(* CoDeSys 2.3.9.62 project: AscensorCompletoDobleV1-2.pro *)
(* Libraries: Standard.lib 2.6.14 10:37:46, IecSfc.lib 2.6.14 12:37:46 *)

(* Global variable list: Global_Variables *)
VAR_GLOBAL
   (*Entradas *)
      (* Sensores de posición en plantas *)
      S0_1: BOOL;
      S1_1: BOOL;
      S2_1: BOOL;
      S3_1: BOOL;
      S0_2: BOOL;
      S1_2: BOOL;
      S2_2: BOOL;
      S3_2: BOOL;
      (* Pulsadores de llamadas en planta *)
      P0: BOOL;
      P1: BOOL;
      P2: BOOL;
      P3: BOOL;
    (* Pulsadores en cabina  *)
      C0_1: BOOL;
      C1_1: BOOL;
      C2_1: BOOL;
      C3_1: BOOL;
      C0_2: BOOL;
      C1_2: BOOL;
      C2_2: BOOL;
      C3_2: BOOL;
   (*Salidas *)
      Motor_arriba_1 : BOOL;
      Motor_Abajo_1 : BOOL;
     Motor_arriba_2 : BOOL;
      Motor_Abajo_2 : BOOL;
   (* luces asociadas a los pulsadores. Se usarán
        si se quiere implementar memoria de llamada *)
     LuzP0:BOOL;
     LuzP1:BOOL;
     LuzP2:BOOL;
     LuzP3:BOOL;
     LuzC0_1:BOOL;
     LuzC1_1:BOOL;
     LuzC2_1:BOOL;
     LuzC3_1:BOOL;
     LuzC0_2:BOOL;
     LuzC1_2:BOOL;
     LuzC2_2:BOOL;
     LuzC3_2:BOOL;
END_VAR

(* POU PLC_PRG, ST *)
PROGRAM PLC_PRG
VAR
	memoria11 : INT := 0;
	memoria12 : INT := 0;
	memoria13 : INT  :=0;
END_VAR
Movimiento1;
Movimiento2;

(* Ascensor 1 *)
Ascensor1;
END_PROGRAM

(* POU Movimiento1, ST *)
PROGRAM Movimiento1
VAR
    pos1:INT:=0;
END_VAR
IF (Motor_arriba_1 AND pos1>=-240) THEN
   pos1:=pos1-2;
END_IF


IF (Motor_abajo_1 AND pos1<=-2) THEN
   pos1:=pos1+2;
END_IF

IF (pos1>=0 AND pos1<=2) THEN
  S0_1:=TRUE;
ELSE
  S0_1:=FALSE;
END_IF

IF (pos1>=-78 AND pos1<=-74) THEN
  S1_1:=TRUE;
ELSE
  S1_1:=FALSE;
END_IF

IF (pos1>=-156 AND pos1<=-152) THEN
  S2_1:=TRUE;
ELSE
  S2_1:=FALSE;
END_IF

IF (pos1>=-242 AND pos1<=-240) THEN
  S3_1:=TRUE;
ELSE
  S3_1:=FALSE;
END_IF
END_PROGRAM

(* POU Movimiento2, ST *)
PROGRAM Movimiento2
VAR
    pos2:INT:=0;
END_VAR
IF (Motor_arriba_2 AND pos2>=-240) THEN
   pos2:=pos2-2;
END_IF


IF (Motor_abajo_2 AND pos2<=-2) THEN
   pos2:=pos2+2;
END_IF

IF (pos2>=0 AND pos2<=2) THEN
  S0_2:=TRUE;
ELSE
  S0_2:=FALSE;
END_IF

IF (pos2>=-78 AND pos2<=-74) THEN
  S1_2:=TRUE;
ELSE
  S1_2:=FALSE;
END_IF

IF (pos2>=-156 AND pos2<=-152) THEN
  S2_2:=TRUE;
ELSE
  S2_2:=FALSE;
END_IF

IF (pos2>=-242 AND pos2<=-240) THEN
  S3_2:=TRUE;
ELSE
  S3_2:=FALSE;
END_IF
END_PROGRAM

(* POU Ascensor1, LD *)
PROGRAM Ascensor1
VAR
	Parado1: BOOL;
	Marcha1: BOOL;
	Sube1_12: BOOL;
	Sube1_01: BOOL;
	Sube1_02: BOOL;
	Sube1_03: BOOL;
	Baja1_10: BOOL;
	Sube1_13: BOOL;
	Baja1_20: BOOL;
	Baja1_21: BOOL;
	Sube1_23: BOOL;
	Baja1_30: BOOL;
	Baja1_31: BOOL;
	Baja1_32: BOOL;
	Marcha2: BOOL;
	Sube2_01: BOOL;
	Sube2_02: BOOL;
	Sube2_03: BOOL;
	Baja2_10: BOOL;
	Sube2_12: BOOL;
	Sube2_13: BOOL;
	Baja2_20: BOOL;
	Baja2_21: BOOL;
	Sube2_23: BOOL;
	Baja2_30: BOOL;
	Baja2_31: BOOL;
	Baja2_32: BOOL;
	FIN: BOOL;
END_VAR
VAR (* helpers for the ST form of the networks *)
	_p1 : BOOL;
	_p2 : BOOL;
	_p3 : BOOL;
	_p4 : BOOL;
	_p5 : BOOL;
	_p6 : BOOL;
	_p7 : BOOL;
	_p8 : BOOL;
	_p9 : BOOL;
	_p10 : BOOL;
	_p11 : BOOL;
	_p12 : BOOL;
	_p13 : BOOL;
	_p14 : BOOL;
	_p15 : BOOL;
	_p16 : BOOL;
	_p17 : BOOL;
	_p18 : BOOL;
	_p19 : BOOL;
	_p20 : BOOL;
	_p21 : BOOL;
	_p22 : BOOL;
	_p23 : BOOL;
	_p24 : BOOL;
	_p25 : BOOL;
	_p26 : BOOL;
	_p27 : BOOL;
	_p28 : BOOL;
	_p29 : BOOL;
	_p30 : BOOL;
	_p31 : BOOL;
	_p32 : BOOL;
	_p33 : BOOL;
	_p34 : BOOL;
	_p35 : BOOL;
	_p36 : BOOL;
	_p37 : BOOL;
	_p38 : BOOL;
	_p39 : BOOL;
	_p40 : BOOL;
	_p41 : BOOL;
	_p42 : BOOL;
	_p43 : BOOL;
	_p44 : BOOL;
	_p45 : BOOL;
	_p46 : BOOL;
	_p47 : BOOL;
	_p48 : BOOL;
	_p49 : BOOL;
	_p50 : BOOL;
	_p51 : BOOL;
	_p52 : BOOL;
	_p53 : BOOL;
	_p54 : BOOL;
	_p55 : BOOL;
	_p56 : BOOL;
	_p57 : BOOL;
	_p58 : BOOL;
	_p59 : BOOL;
	_p60 : BOOL;
	_p61 : BOOL;
	_p62 : BOOL;
END_VAR
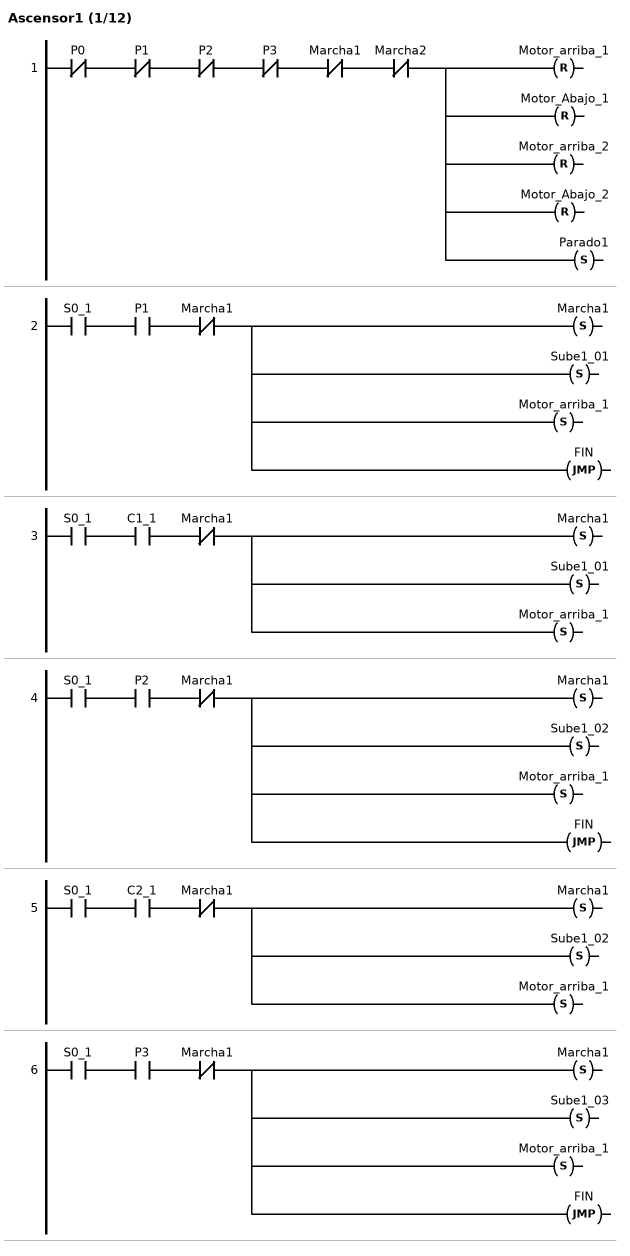
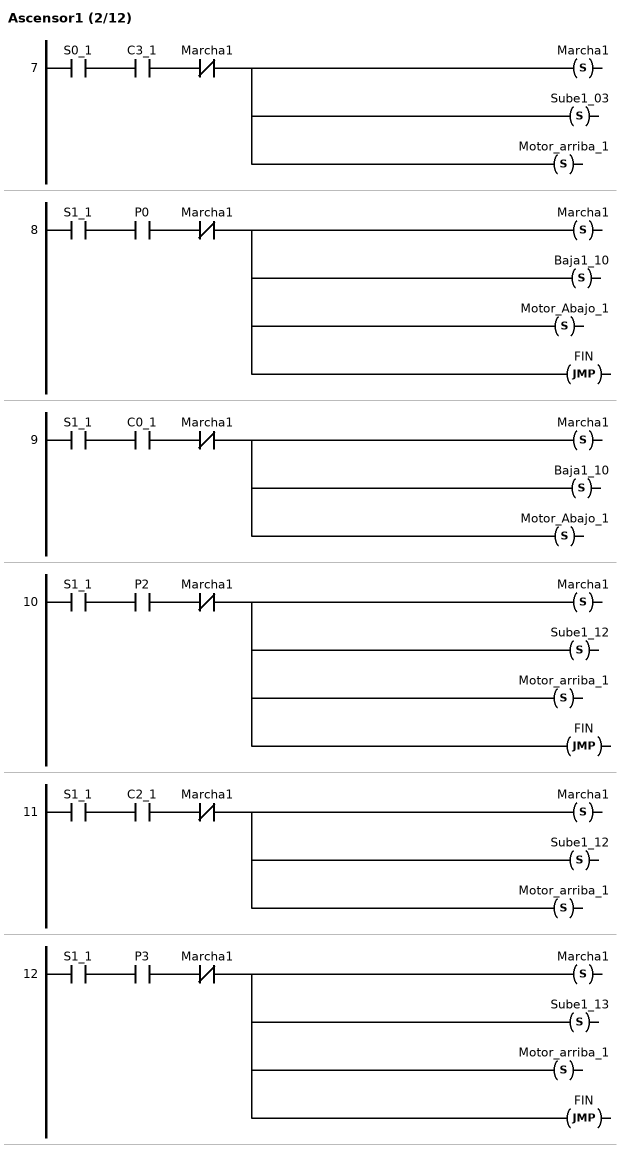
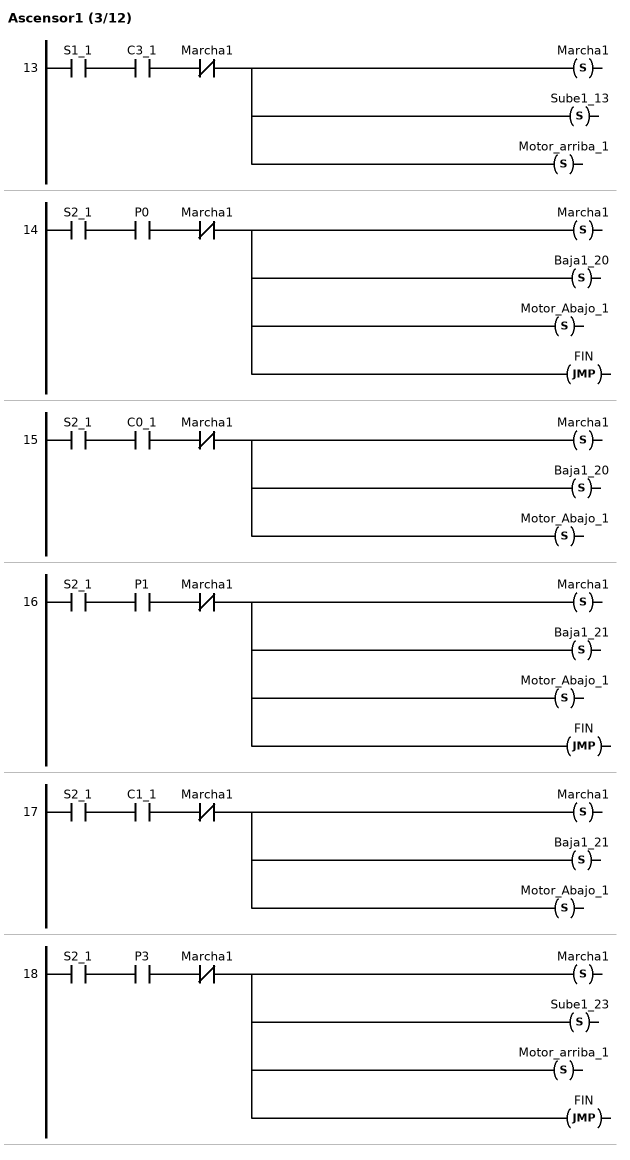
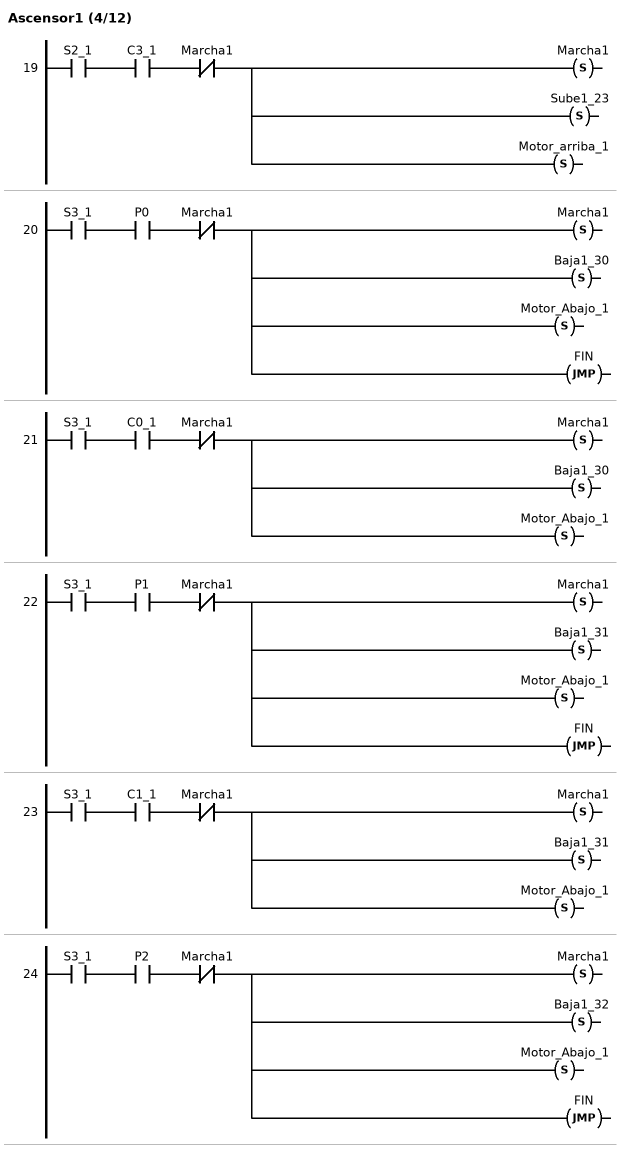
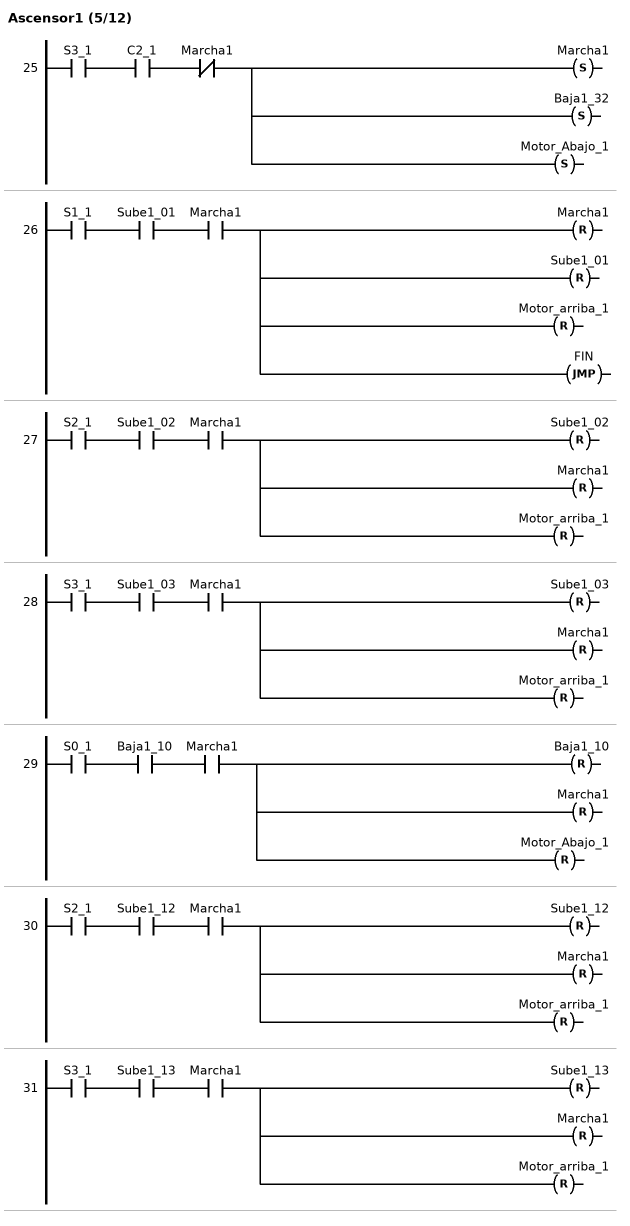
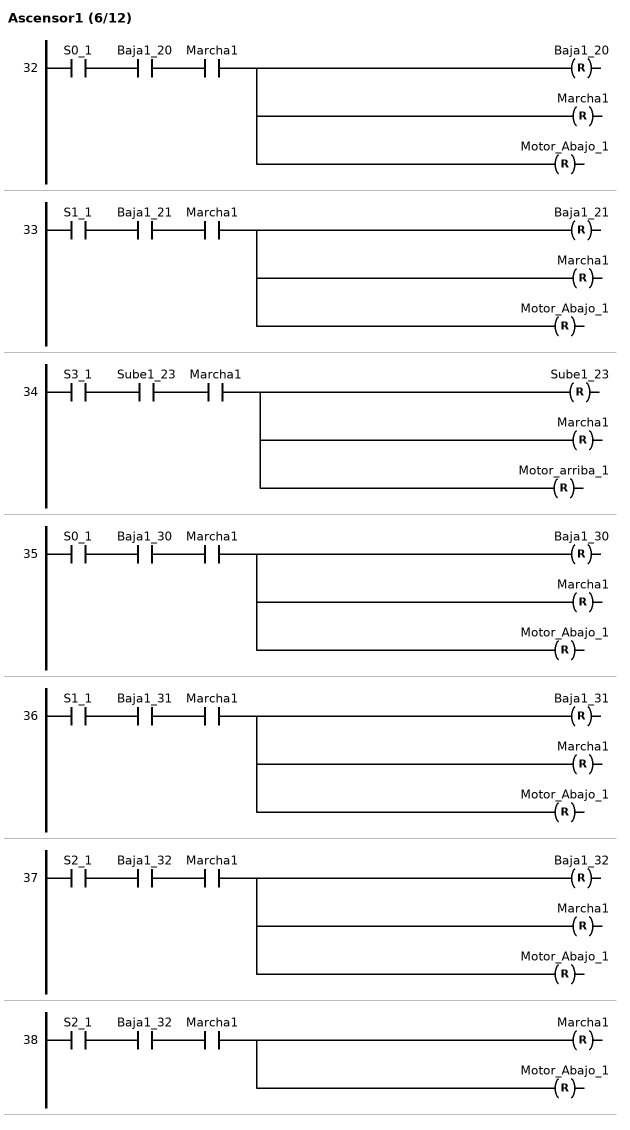
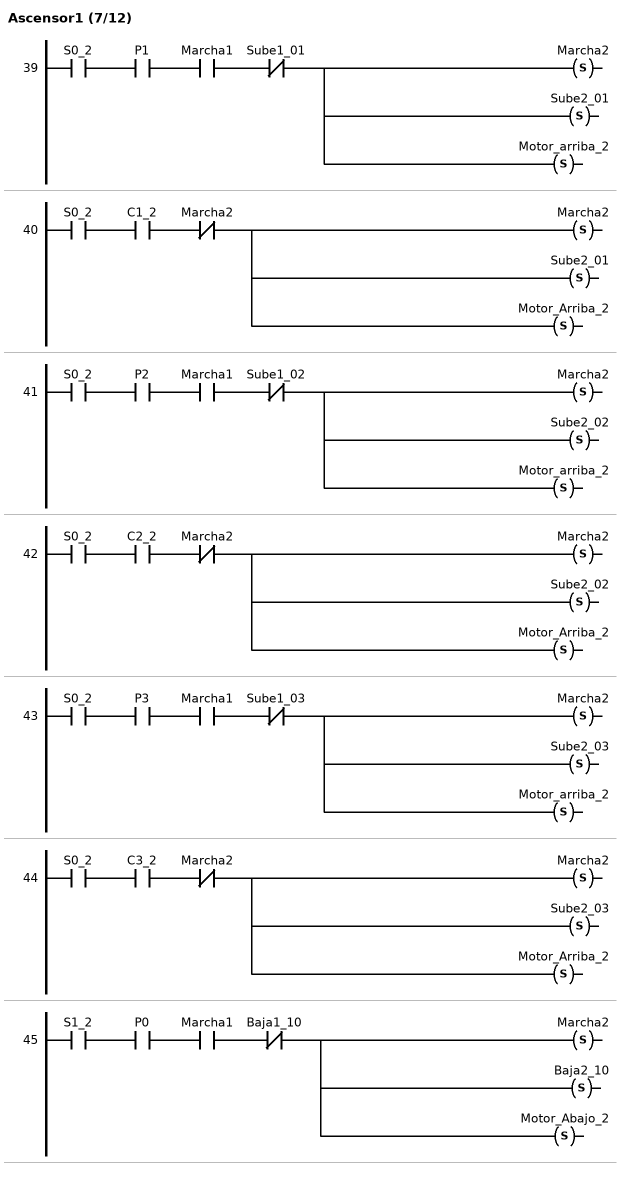
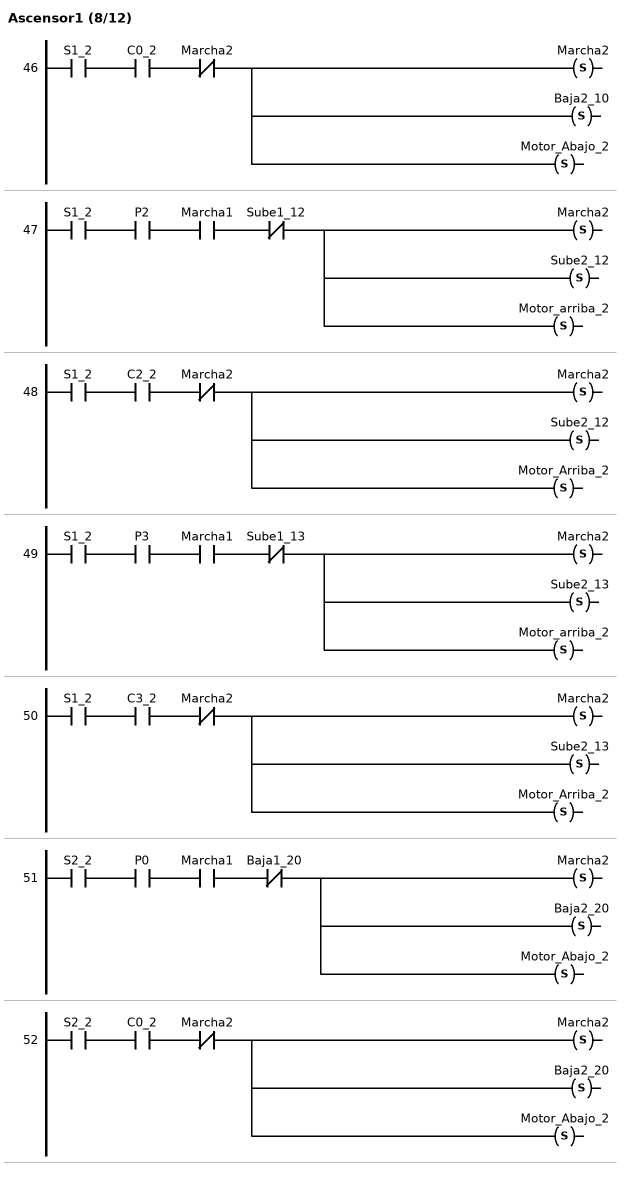
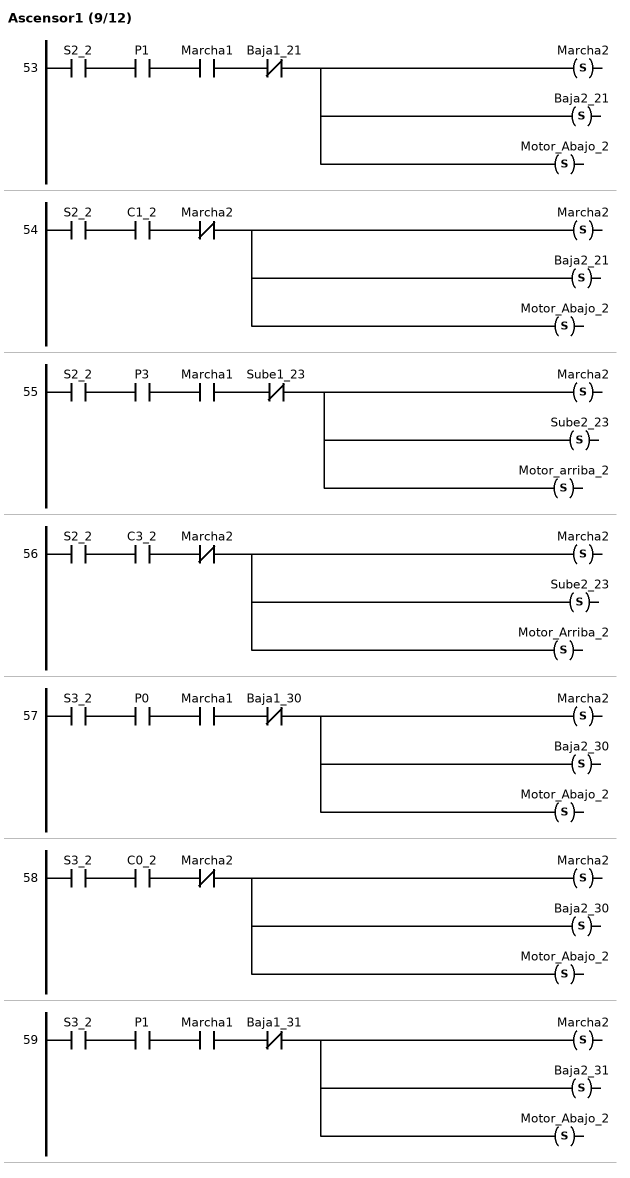
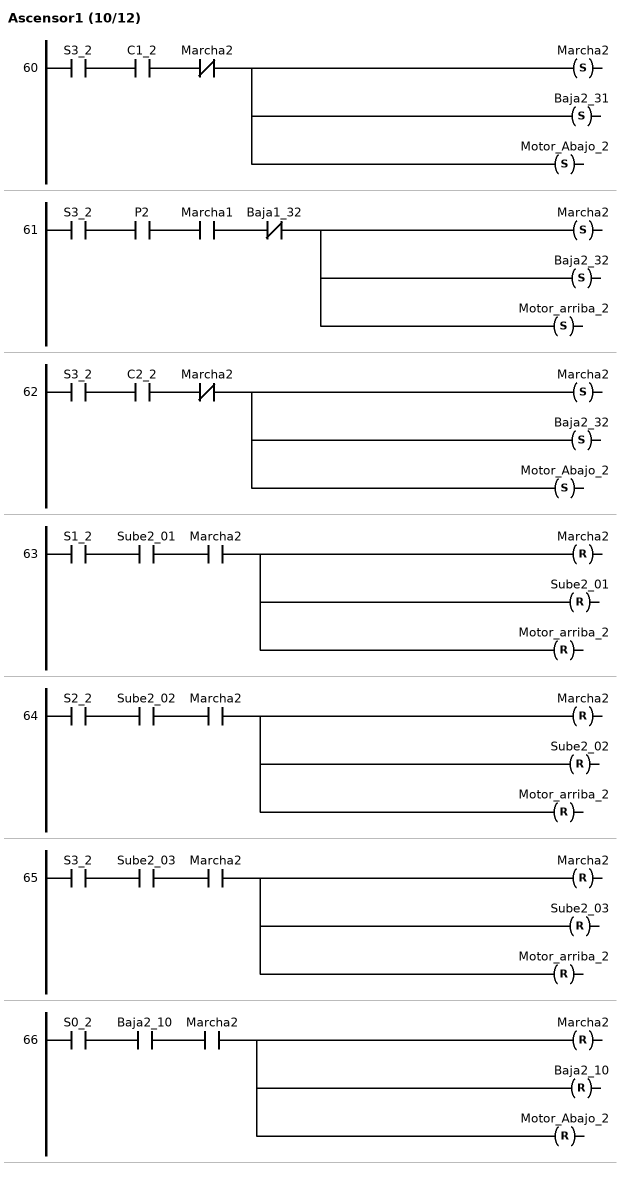
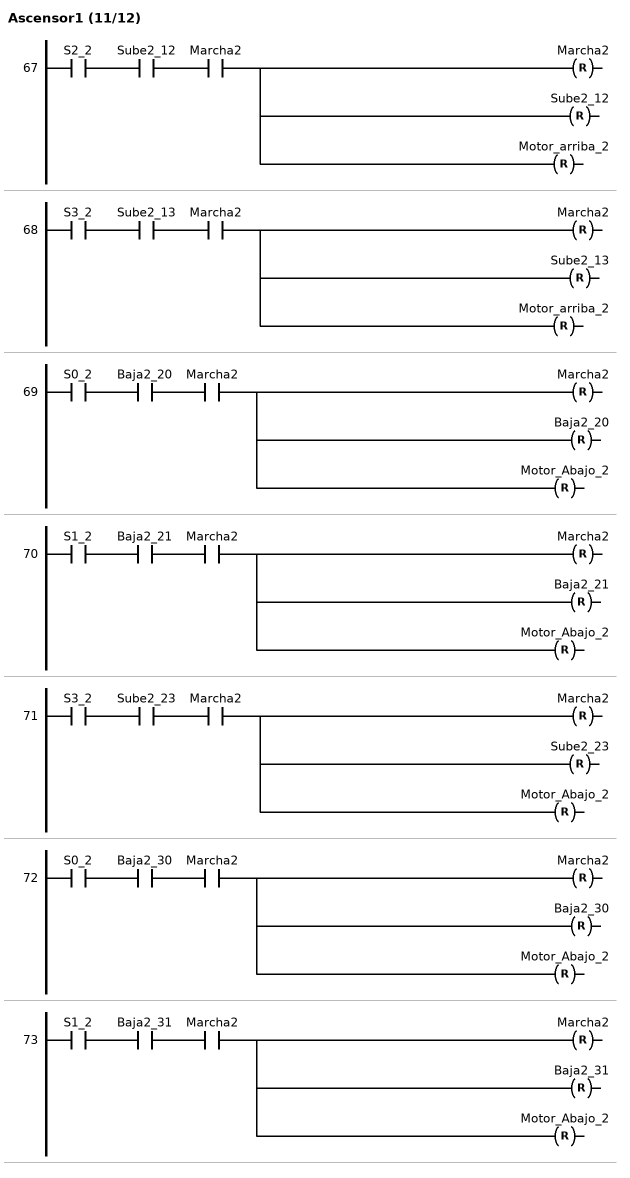
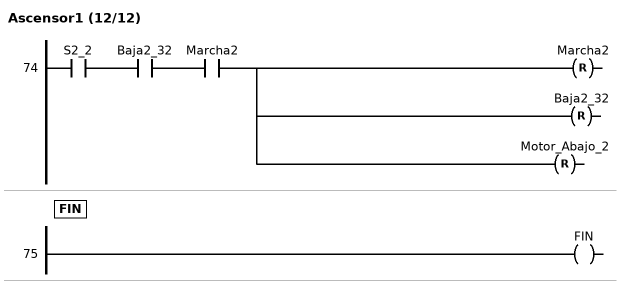
_LD_ (* Ladder Diagram *)
NETWORK 1
	[/P0] - [/P1] - [/P2] - [/P3] - [/Marcha1] - [/Marcha2] --- (R Motor_arriba_1) (R Motor_Abajo_1) (R Motor_arriba_2) (R Motor_Abajo_2) (S Parado1)
NETWORK 2
	[S0_1] - [P1] - [/Marcha1] --- (S Marcha1) (S Sube1_01) (S Motor_arriba_1) >>FIN
NETWORK 3
	[S0_1] - [C1_1] - [/Marcha1] --- (S Marcha1) (S Sube1_01) (S Motor_arriba_1)
NETWORK 4
	[S0_1] - [P2] - [/Marcha1] --- (S Marcha1) (S Sube1_02) (S Motor_arriba_1) >>FIN
NETWORK 5
	[S0_1] - [C2_1] - [/Marcha1] --- (S Marcha1) (S Sube1_02) (S Motor_arriba_1)
NETWORK 6
	[S0_1] - [P3] - [/Marcha1] --- (S Marcha1) (S Sube1_03) (S Motor_arriba_1) >>FIN
NETWORK 7
	[S0_1] - [C3_1] - [/Marcha1] --- (S Marcha1) (S Sube1_03) (S Motor_arriba_1)
NETWORK 8
	[S1_1] - [P0] - [/Marcha1] --- (S Marcha1) (S Baja1_10) (S Motor_Abajo_1) >>FIN
NETWORK 9
	[S1_1] - [C0_1] - [/Marcha1] --- (S Marcha1) (S Baja1_10) (S Motor_Abajo_1)
NETWORK 10
	[S1_1] - [P2] - [/Marcha1] --- (S Marcha1) (S Sube1_12) (S Motor_arriba_1) >>FIN
NETWORK 11
	[S1_1] - [C2_1] - [/Marcha1] --- (S Marcha1) (S Sube1_12) (S Motor_arriba_1)
NETWORK 12
	[S1_1] - [P3] - [/Marcha1] --- (S Marcha1) (S Sube1_13) (S Motor_arriba_1) >>FIN
NETWORK 13
	[S1_1] - [C3_1] - [/Marcha1] --- (S Marcha1) (S Sube1_13) (S Motor_arriba_1)
NETWORK 14
	[S2_1] - [P0] - [/Marcha1] --- (S Marcha1) (S Baja1_20) (S Motor_Abajo_1) >>FIN
NETWORK 15
	[S2_1] - [C0_1] - [/Marcha1] --- (S Marcha1) (S Baja1_20) (S Motor_Abajo_1)
NETWORK 16
	[S2_1] - [P1] - [/Marcha1] --- (S Marcha1) (S Baja1_21) (S Motor_Abajo_1) >>FIN
NETWORK 17
	[S2_1] - [C1_1] - [/Marcha1] --- (S Marcha1) (S Baja1_21) (S Motor_Abajo_1)
NETWORK 18
	[S2_1] - [P3] - [/Marcha1] --- (S Marcha1) (S Sube1_23) (S Motor_arriba_1) >>FIN
NETWORK 19
	[S2_1] - [C3_1] - [/Marcha1] --- (S Marcha1) (S Sube1_23) (S Motor_arriba_1)
NETWORK 20
	[S3_1] - [P0] - [/Marcha1] --- (S Marcha1) (S Baja1_30) (S Motor_Abajo_1) >>FIN
NETWORK 21
	[S3_1] - [C0_1] - [/Marcha1] --- (S Marcha1) (S Baja1_30) (S Motor_Abajo_1)
NETWORK 22
	[S3_1] - [P1] - [/Marcha1] --- (S Marcha1) (S Baja1_31) (S Motor_Abajo_1) >>FIN
NETWORK 23
	[S3_1] - [C1_1] - [/Marcha1] --- (S Marcha1) (S Baja1_31) (S Motor_Abajo_1)
NETWORK 24
	[S3_1] - [P2] - [/Marcha1] --- (S Marcha1) (S Baja1_32) (S Motor_Abajo_1) >>FIN
NETWORK 25
	[S3_1] - [C2_1] - [/Marcha1] --- (S Marcha1) (S Baja1_32) (S Motor_Abajo_1)
NETWORK 26
	[S1_1] - [Sube1_01] - [Marcha1] --- (R Marcha1) (R Sube1_01) (R Motor_arriba_1) >>FIN
NETWORK 27
	[S2_1] - [Sube1_02] - [Marcha1] --- (R Sube1_02) (R Marcha1) (R Motor_arriba_1)
NETWORK 28
	[S3_1] - [Sube1_03] - [Marcha1] --- (R Sube1_03) (R Marcha1) (R Motor_arriba_1)
NETWORK 29
	[S0_1] - [Baja1_10] - [Marcha1] --- (R Baja1_10) (R Marcha1) (R Motor_Abajo_1)
NETWORK 30
	[S2_1] - [Sube1_12] - [Marcha1] --- (R Sube1_12) (R Marcha1) (R Motor_arriba_1)
NETWORK 31
	[S3_1] - [Sube1_13] - [Marcha1] --- (R Sube1_13) (R Marcha1) (R Motor_arriba_1)
NETWORK 32
	[S0_1] - [Baja1_20] - [Marcha1] --- (R Baja1_20) (R Marcha1) (R Motor_Abajo_1)
NETWORK 33
	[S1_1] - [Baja1_21] - [Marcha1] --- (R Baja1_21) (R Marcha1) (R Motor_Abajo_1)
NETWORK 34
	[S3_1] - [Sube1_23] - [Marcha1] --- (R Sube1_23) (R Marcha1) (R Motor_arriba_1)
NETWORK 35
	[S0_1] - [Baja1_30] - [Marcha1] --- (R Baja1_30) (R Marcha1) (R Motor_Abajo_1)
NETWORK 36
	[S1_1] - [Baja1_31] - [Marcha1] --- (R Baja1_31) (R Marcha1) (R Motor_Abajo_1)
NETWORK 37
	[S2_1] - [Baja1_32] - [Marcha1] --- (R Baja1_32) (R Marcha1) (R Motor_Abajo_1)
NETWORK 38
	[S2_1] - [Baja1_32] - [Marcha1] --- (R Marcha1) (R Motor_Abajo_1)
NETWORK 39
	[S0_2] - [P1] - [Marcha1] - [/Sube1_01] --- (S Marcha2) (S Sube2_01) (S Motor_arriba_2)
NETWORK 40
	[S0_2] - [C1_2] - [/Marcha2] --- (S Marcha2) (S Sube2_01) (S Motor_Arriba_2)
NETWORK 41
	[S0_2] - [P2] - [Marcha1] - [/Sube1_02] --- (S Marcha2) (S Sube2_02) (S Motor_arriba_2)
NETWORK 42
	[S0_2] - [C2_2] - [/Marcha2] --- (S Marcha2) (S Sube2_02) (S Motor_Arriba_2)
NETWORK 43
	[S0_2] - [P3] - [Marcha1] - [/Sube1_03] --- (S Marcha2) (S Sube2_03) (S Motor_arriba_2)
NETWORK 44
	[S0_2] - [C3_2] - [/Marcha2] --- (S Marcha2) (S Sube2_03) (S Motor_Arriba_2)
NETWORK 45
	[S1_2] - [P0] - [Marcha1] - [/Baja1_10] --- (S Marcha2) (S Baja2_10) (S Motor_Abajo_2)
NETWORK 46
	[S1_2] - [C0_2] - [/Marcha2] --- (S Marcha2) (S Baja2_10) (S Motor_Abajo_2)
NETWORK 47
	[S1_2] - [P2] - [Marcha1] - [/Sube1_12] --- (S Marcha2) (S Sube2_12) (S Motor_arriba_2)
NETWORK 48
	[S1_2] - [C2_2] - [/Marcha2] --- (S Marcha2) (S Sube2_12) (S Motor_Arriba_2)
NETWORK 49
	[S1_2] - [P3] - [Marcha1] - [/Sube1_13] --- (S Marcha2) (S Sube2_13) (S Motor_arriba_2)
NETWORK 50
	[S1_2] - [C3_2] - [/Marcha2] --- (S Marcha2) (S Sube2_13) (S Motor_Arriba_2)
NETWORK 51
	[S2_2] - [P0] - [Marcha1] - [/Baja1_20] --- (S Marcha2) (S Baja2_20) (S Motor_Abajo_2)
NETWORK 52
	[S2_2] - [C0_2] - [/Marcha2] --- (S Marcha2) (S Baja2_20) (S Motor_Abajo_2)
NETWORK 53
	[S2_2] - [P1] - [Marcha1] - [/Baja1_21] --- (S Marcha2) (S Baja2_21) (S Motor_Abajo_2)
NETWORK 54
	[S2_2] - [C1_2] - [/Marcha2] --- (S Marcha2) (S Baja2_21) (S Motor_Abajo_2)
NETWORK 55
	[S2_2] - [P3] - [Marcha1] - [/Sube1_23] --- (S Marcha2) (S Sube2_23) (S Motor_arriba_2)
NETWORK 56
	[S2_2] - [C3_2] - [/Marcha2] --- (S Marcha2) (S Sube2_23) (S Motor_Arriba_2)
NETWORK 57
	[S3_2] - [P0] - [Marcha1] - [/Baja1_30] --- (S Marcha2) (S Baja2_30) (S Motor_Abajo_2)
NETWORK 58
	[S3_2] - [C0_2] - [/Marcha2] --- (S Marcha2) (S Baja2_30) (S Motor_Abajo_2)
NETWORK 59
	[S3_2] - [P1] - [Marcha1] - [/Baja1_31] --- (S Marcha2) (S Baja2_31) (S Motor_Abajo_2)
NETWORK 60
	[S3_2] - [C1_2] - [/Marcha2] --- (S Marcha2) (S Baja2_31) (S Motor_Abajo_2)
NETWORK 61
	[S3_2] - [P2] - [Marcha1] - [/Baja1_32] --- (S Marcha2) (S Baja2_32) (S Motor_arriba_2)
NETWORK 62
	[S3_2] - [C2_2] - [/Marcha2] --- (S Marcha2) (S Baja2_32) (S Motor_Abajo_2)
NETWORK 63
	[S1_2] - [Sube2_01] - [Marcha2] --- (R Marcha2) (R Sube2_01) (R Motor_arriba_2)
NETWORK 64
	[S2_2] - [Sube2_02] - [Marcha2] --- (R Marcha2) (R Sube2_02) (R Motor_arriba_2)
NETWORK 65
	[S3_2] - [Sube2_03] - [Marcha2] --- (R Marcha2) (R Sube2_03) (R Motor_arriba_2)
NETWORK 66
	[S0_2] - [Baja2_10] - [Marcha2] --- (R Marcha2) (R Baja2_10) (R Motor_Abajo_2)
NETWORK 67
	[S2_2] - [Sube2_12] - [Marcha2] --- (R Marcha2) (R Sube2_12) (R Motor_arriba_2)
NETWORK 68
	[S3_2] - [Sube2_13] - [Marcha2] --- (R Marcha2) (R Sube2_13) (R Motor_arriba_2)
NETWORK 69
	[S0_2] - [Baja2_20] - [Marcha2] --- (R Marcha2) (R Baja2_20) (R Motor_Abajo_2)
NETWORK 70
	[S1_2] - [Baja2_21] - [Marcha2] --- (R Marcha2) (R Baja2_21) (R Motor_Abajo_2)
NETWORK 71
	[S3_2] - [Sube2_23] - [Marcha2] --- (R Marcha2) (R Sube2_23) (R Motor_Abajo_2)
NETWORK 72
	[S0_2] - [Baja2_30] - [Marcha2] --- (R Marcha2) (R Baja2_30) (R Motor_Abajo_2)
NETWORK 73
	[S1_2] - [Baja2_31] - [Marcha2] --- (R Marcha2) (R Baja2_31) (R Motor_Abajo_2)
NETWORK 74
	[S2_2] - [Baja2_32] - [Marcha2] --- (R Marcha2) (R Baja2_32) (R Motor_Abajo_2)
NETWORK 75 FIN:
	* --- (FIN)
_END_LD_
(* the same logic as Structured Text *)
(* Network 1 *)
_p1 := NOT P0 AND NOT P1 AND NOT P2 AND NOT P3 AND NOT Marcha1 AND NOT Marcha2;
IF _p1 THEN Motor_arriba_1 := FALSE; Motor_Abajo_1 := FALSE; Motor_arriba_2 := FALSE; Motor_Abajo_2 := FALSE; Parado1 := TRUE; END_IF;
(* Network 2 *)
_p2 := S0_1 AND P1 AND NOT Marcha1;
IF _p2 THEN Marcha1 := TRUE; END_IF;
IF _p2 THEN Sube1_01 := TRUE; END_IF;
IF _p2 THEN Motor_arriba_1 := TRUE; END_IF;
IF _p2 THEN JMP FIN; END_IF;
(* Network 3 *)
_p3 := S0_1 AND C1_1 AND NOT Marcha1;
IF _p3 THEN Marcha1 := TRUE; Sube1_01 := TRUE; Motor_arriba_1 := TRUE; END_IF;
(* Network 4 *)
_p4 := S0_1 AND P2 AND NOT Marcha1;
IF _p4 THEN Marcha1 := TRUE; END_IF;
IF _p4 THEN Sube1_02 := TRUE; END_IF;
IF _p4 THEN Motor_arriba_1 := TRUE; END_IF;
IF _p4 THEN JMP FIN; END_IF;
(* Network 5 *)
_p5 := S0_1 AND C2_1 AND NOT Marcha1;
IF _p5 THEN Marcha1 := TRUE; Sube1_02 := TRUE; Motor_arriba_1 := TRUE; END_IF;
(* Network 6 *)
_p6 := S0_1 AND P3 AND NOT Marcha1;
IF _p6 THEN Marcha1 := TRUE; END_IF;
IF _p6 THEN Sube1_03 := TRUE; END_IF;
IF _p6 THEN Motor_arriba_1 := TRUE; END_IF;
IF _p6 THEN JMP FIN; END_IF;
(* Network 7 *)
_p7 := S0_1 AND C3_1 AND NOT Marcha1;
IF _p7 THEN Marcha1 := TRUE; Sube1_03 := TRUE; Motor_arriba_1 := TRUE; END_IF;
(* Network 8 *)
_p8 := S1_1 AND P0 AND NOT Marcha1;
IF _p8 THEN Marcha1 := TRUE; END_IF;
IF _p8 THEN Baja1_10 := TRUE; END_IF;
IF _p8 THEN Motor_Abajo_1 := TRUE; END_IF;
IF _p8 THEN JMP FIN; END_IF;
(* Network 9 *)
_p9 := S1_1 AND C0_1 AND NOT Marcha1;
IF _p9 THEN Marcha1 := TRUE; Baja1_10 := TRUE; Motor_Abajo_1 := TRUE; END_IF;
(* Network 10 *)
_p10 := S1_1 AND P2 AND NOT Marcha1;
IF _p10 THEN Marcha1 := TRUE; END_IF;
IF _p10 THEN Sube1_12 := TRUE; END_IF;
IF _p10 THEN Motor_arriba_1 := TRUE; END_IF;
IF _p10 THEN JMP FIN; END_IF;
(* Network 11 *)
_p11 := S1_1 AND C2_1 AND NOT Marcha1;
IF _p11 THEN Marcha1 := TRUE; Sube1_12 := TRUE; Motor_arriba_1 := TRUE; END_IF;
(* Network 12 *)
_p12 := S1_1 AND P3 AND NOT Marcha1;
IF _p12 THEN Marcha1 := TRUE; END_IF;
IF _p12 THEN Sube1_13 := TRUE; END_IF;
IF _p12 THEN Motor_arriba_1 := TRUE; END_IF;
IF _p12 THEN JMP FIN; END_IF;
(* Network 13 *)
_p13 := S1_1 AND C3_1 AND NOT Marcha1;
IF _p13 THEN Marcha1 := TRUE; Sube1_13 := TRUE; Motor_arriba_1 := TRUE; END_IF;
(* Network 14 *)
_p14 := S2_1 AND P0 AND NOT Marcha1;
IF _p14 THEN Marcha1 := TRUE; END_IF;
IF _p14 THEN Baja1_20 := TRUE; END_IF;
IF _p14 THEN Motor_Abajo_1 := TRUE; END_IF;
IF _p14 THEN JMP FIN; END_IF;
(* Network 15 *)
_p15 := S2_1 AND C0_1 AND NOT Marcha1;
IF _p15 THEN Marcha1 := TRUE; Baja1_20 := TRUE; Motor_Abajo_1 := TRUE; END_IF;
(* Network 16 *)
_p16 := S2_1 AND P1 AND NOT Marcha1;
IF _p16 THEN Marcha1 := TRUE; END_IF;
IF _p16 THEN Baja1_21 := TRUE; END_IF;
IF _p16 THEN Motor_Abajo_1 := TRUE; END_IF;
IF _p16 THEN JMP FIN; END_IF;
(* Network 17 *)
_p17 := S2_1 AND C1_1 AND NOT Marcha1;
IF _p17 THEN Marcha1 := TRUE; Baja1_21 := TRUE; Motor_Abajo_1 := TRUE; END_IF;
(* Network 18 *)
_p18 := S2_1 AND P3 AND NOT Marcha1;
IF _p18 THEN Marcha1 := TRUE; END_IF;
IF _p18 THEN Sube1_23 := TRUE; END_IF;
IF _p18 THEN Motor_arriba_1 := TRUE; END_IF;
IF _p18 THEN JMP FIN; END_IF;
(* Network 19 *)
_p19 := S2_1 AND C3_1 AND NOT Marcha1;
IF _p19 THEN Marcha1 := TRUE; Sube1_23 := TRUE; Motor_arriba_1 := TRUE; END_IF;
(* Network 20 *)
_p20 := S3_1 AND P0 AND NOT Marcha1;
IF _p20 THEN Marcha1 := TRUE; END_IF;
IF _p20 THEN Baja1_30 := TRUE; END_IF;
IF _p20 THEN Motor_Abajo_1 := TRUE; END_IF;
IF _p20 THEN JMP FIN; END_IF;
(* Network 21 *)
_p21 := S3_1 AND C0_1 AND NOT Marcha1;
IF _p21 THEN Marcha1 := TRUE; Baja1_30 := TRUE; Motor_Abajo_1 := TRUE; END_IF;
(* Network 22 *)
_p22 := S3_1 AND P1 AND NOT Marcha1;
IF _p22 THEN Marcha1 := TRUE; END_IF;
IF _p22 THEN Baja1_31 := TRUE; END_IF;
IF _p22 THEN Motor_Abajo_1 := TRUE; END_IF;
IF _p22 THEN JMP FIN; END_IF;
(* Network 23 *)
_p23 := S3_1 AND C1_1 AND NOT Marcha1;
IF _p23 THEN Marcha1 := TRUE; Baja1_31 := TRUE; Motor_Abajo_1 := TRUE; END_IF;
(* Network 24 *)
_p24 := S3_1 AND P2 AND NOT Marcha1;
IF _p24 THEN Marcha1 := TRUE; END_IF;
IF _p24 THEN Baja1_32 := TRUE; END_IF;
IF _p24 THEN Motor_Abajo_1 := TRUE; END_IF;
IF _p24 THEN JMP FIN; END_IF;
(* Network 25 *)
_p25 := S3_1 AND C2_1 AND NOT Marcha1;
IF _p25 THEN Marcha1 := TRUE; Baja1_32 := TRUE; Motor_Abajo_1 := TRUE; END_IF;
(* Network 26 *)
_p26 := S1_1 AND Sube1_01 AND Marcha1;
IF _p26 THEN Marcha1 := FALSE; END_IF;
IF _p26 THEN Sube1_01 := FALSE; END_IF;
IF _p26 THEN Motor_arriba_1 := FALSE; END_IF;
IF _p26 THEN JMP FIN; END_IF;
(* Network 27 *)
_p27 := S2_1 AND Sube1_02 AND Marcha1;
IF _p27 THEN Sube1_02 := FALSE; Marcha1 := FALSE; Motor_arriba_1 := FALSE; END_IF;
(* Network 28 *)
_p28 := S3_1 AND Sube1_03 AND Marcha1;
IF _p28 THEN Sube1_03 := FALSE; Marcha1 := FALSE; Motor_arriba_1 := FALSE; END_IF;
(* Network 29 *)
_p29 := S0_1 AND Baja1_10 AND Marcha1;
IF _p29 THEN Baja1_10 := FALSE; Marcha1 := FALSE; Motor_Abajo_1 := FALSE; END_IF;
(* Network 30 *)
_p30 := S2_1 AND Sube1_12 AND Marcha1;
IF _p30 THEN Sube1_12 := FALSE; Marcha1 := FALSE; Motor_arriba_1 := FALSE; END_IF;
(* Network 31 *)
_p31 := S3_1 AND Sube1_13 AND Marcha1;
IF _p31 THEN Sube1_13 := FALSE; Marcha1 := FALSE; Motor_arriba_1 := FALSE; END_IF;
(* Network 32 *)
_p32 := S0_1 AND Baja1_20 AND Marcha1;
IF _p32 THEN Baja1_20 := FALSE; Marcha1 := FALSE; Motor_Abajo_1 := FALSE; END_IF;
(* Network 33 *)
_p33 := S1_1 AND Baja1_21 AND Marcha1;
IF _p33 THEN Baja1_21 := FALSE; Marcha1 := FALSE; Motor_Abajo_1 := FALSE; END_IF;
(* Network 34 *)
_p34 := S3_1 AND Sube1_23 AND Marcha1;
IF _p34 THEN Sube1_23 := FALSE; Marcha1 := FALSE; Motor_arriba_1 := FALSE; END_IF;
(* Network 35 *)
_p35 := S0_1 AND Baja1_30 AND Marcha1;
IF _p35 THEN Baja1_30 := FALSE; Marcha1 := FALSE; Motor_Abajo_1 := FALSE; END_IF;
(* Network 36 *)
_p36 := S1_1 AND Baja1_31 AND Marcha1;
IF _p36 THEN Baja1_31 := FALSE; Marcha1 := FALSE; Motor_Abajo_1 := FALSE; END_IF;
(* Network 37 *)
_p37 := S2_1 AND Baja1_32 AND Marcha1;
IF _p37 THEN Baja1_32 := FALSE; Marcha1 := FALSE; Motor_Abajo_1 := FALSE; END_IF;
(* Network 38 *)
_p38 := S2_1 AND Baja1_32 AND Marcha1;
IF _p38 THEN Marcha1 := FALSE; Motor_Abajo_1 := FALSE; END_IF;
(* Network 39 *)
IF S0_2 AND P1 AND Marcha1 AND NOT Sube1_01 THEN Marcha2 := TRUE; Sube2_01 := TRUE; Motor_arriba_2 := TRUE; END_IF;
(* Network 40 *)
_p39 := S0_2 AND C1_2 AND NOT Marcha2;
IF _p39 THEN Marcha2 := TRUE; Sube2_01 := TRUE; Motor_Arriba_2 := TRUE; END_IF;
(* Network 41 *)
IF S0_2 AND P2 AND Marcha1 AND NOT Sube1_02 THEN Marcha2 := TRUE; Sube2_02 := TRUE; Motor_arriba_2 := TRUE; END_IF;
(* Network 42 *)
_p40 := S0_2 AND C2_2 AND NOT Marcha2;
IF _p40 THEN Marcha2 := TRUE; Sube2_02 := TRUE; Motor_Arriba_2 := TRUE; END_IF;
(* Network 43 *)
IF S0_2 AND P3 AND Marcha1 AND NOT Sube1_03 THEN Marcha2 := TRUE; Sube2_03 := TRUE; Motor_arriba_2 := TRUE; END_IF;
(* Network 44 *)
_p41 := S0_2 AND C3_2 AND NOT Marcha2;
IF _p41 THEN Marcha2 := TRUE; Sube2_03 := TRUE; Motor_Arriba_2 := TRUE; END_IF;
(* Network 45 *)
IF S1_2 AND P0 AND Marcha1 AND NOT Baja1_10 THEN Marcha2 := TRUE; Baja2_10 := TRUE; Motor_Abajo_2 := TRUE; END_IF;
(* Network 46 *)
_p42 := S1_2 AND C0_2 AND NOT Marcha2;
IF _p42 THEN Marcha2 := TRUE; Baja2_10 := TRUE; Motor_Abajo_2 := TRUE; END_IF;
(* Network 47 *)
IF S1_2 AND P2 AND Marcha1 AND NOT Sube1_12 THEN Marcha2 := TRUE; Sube2_12 := TRUE; Motor_arriba_2 := TRUE; END_IF;
(* Network 48 *)
_p43 := S1_2 AND C2_2 AND NOT Marcha2;
IF _p43 THEN Marcha2 := TRUE; Sube2_12 := TRUE; Motor_Arriba_2 := TRUE; END_IF;
(* Network 49 *)
IF S1_2 AND P3 AND Marcha1 AND NOT Sube1_13 THEN Marcha2 := TRUE; Sube2_13 := TRUE; Motor_arriba_2 := TRUE; END_IF;
(* Network 50 *)
_p44 := S1_2 AND C3_2 AND NOT Marcha2;
IF _p44 THEN Marcha2 := TRUE; Sube2_13 := TRUE; Motor_Arriba_2 := TRUE; END_IF;
(* Network 51 *)
IF S2_2 AND P0 AND Marcha1 AND NOT Baja1_20 THEN Marcha2 := TRUE; Baja2_20 := TRUE; Motor_Abajo_2 := TRUE; END_IF;
(* Network 52 *)
_p45 := S2_2 AND C0_2 AND NOT Marcha2;
IF _p45 THEN Marcha2 := TRUE; Baja2_20 := TRUE; Motor_Abajo_2 := TRUE; END_IF;
(* Network 53 *)
IF S2_2 AND P1 AND Marcha1 AND NOT Baja1_21 THEN Marcha2 := TRUE; Baja2_21 := TRUE; Motor_Abajo_2 := TRUE; END_IF;
(* Network 54 *)
_p46 := S2_2 AND C1_2 AND NOT Marcha2;
IF _p46 THEN Marcha2 := TRUE; Baja2_21 := TRUE; Motor_Abajo_2 := TRUE; END_IF;
(* Network 55 *)
IF S2_2 AND P3 AND Marcha1 AND NOT Sube1_23 THEN Marcha2 := TRUE; Sube2_23 := TRUE; Motor_arriba_2 := TRUE; END_IF;
(* Network 56 *)
_p47 := S2_2 AND C3_2 AND NOT Marcha2;
IF _p47 THEN Marcha2 := TRUE; Sube2_23 := TRUE; Motor_Arriba_2 := TRUE; END_IF;
(* Network 57 *)
IF S3_2 AND P0 AND Marcha1 AND NOT Baja1_30 THEN Marcha2 := TRUE; Baja2_30 := TRUE; Motor_Abajo_2 := TRUE; END_IF;
(* Network 58 *)
_p48 := S3_2 AND C0_2 AND NOT Marcha2;
IF _p48 THEN Marcha2 := TRUE; Baja2_30 := TRUE; Motor_Abajo_2 := TRUE; END_IF;
(* Network 59 *)
IF S3_2 AND P1 AND Marcha1 AND NOT Baja1_31 THEN Marcha2 := TRUE; Baja2_31 := TRUE; Motor_Abajo_2 := TRUE; END_IF;
(* Network 60 *)
_p49 := S3_2 AND C1_2 AND NOT Marcha2;
IF _p49 THEN Marcha2 := TRUE; Baja2_31 := TRUE; Motor_Abajo_2 := TRUE; END_IF;
(* Network 61 *)
IF S3_2 AND P2 AND Marcha1 AND NOT Baja1_32 THEN Marcha2 := TRUE; Baja2_32 := TRUE; Motor_arriba_2 := TRUE; END_IF;
(* Network 62 *)
_p50 := S3_2 AND C2_2 AND NOT Marcha2;
IF _p50 THEN Marcha2 := TRUE; Baja2_32 := TRUE; Motor_Abajo_2 := TRUE; END_IF;
(* Network 63 *)
_p51 := S1_2 AND Sube2_01 AND Marcha2;
IF _p51 THEN Marcha2 := FALSE; Sube2_01 := FALSE; Motor_arriba_2 := FALSE; END_IF;
(* Network 64 *)
_p52 := S2_2 AND Sube2_02 AND Marcha2;
IF _p52 THEN Marcha2 := FALSE; Sube2_02 := FALSE; Motor_arriba_2 := FALSE; END_IF;
(* Network 65 *)
_p53 := S3_2 AND Sube2_03 AND Marcha2;
IF _p53 THEN Marcha2 := FALSE; Sube2_03 := FALSE; Motor_arriba_2 := FALSE; END_IF;
(* Network 66 *)
_p54 := S0_2 AND Baja2_10 AND Marcha2;
IF _p54 THEN Marcha2 := FALSE; Baja2_10 := FALSE; Motor_Abajo_2 := FALSE; END_IF;
(* Network 67 *)
_p55 := S2_2 AND Sube2_12 AND Marcha2;
IF _p55 THEN Marcha2 := FALSE; Sube2_12 := FALSE; Motor_arriba_2 := FALSE; END_IF;
(* Network 68 *)
_p56 := S3_2 AND Sube2_13 AND Marcha2;
IF _p56 THEN Marcha2 := FALSE; Sube2_13 := FALSE; Motor_arriba_2 := FALSE; END_IF;
(* Network 69 *)
_p57 := S0_2 AND Baja2_20 AND Marcha2;
IF _p57 THEN Marcha2 := FALSE; Baja2_20 := FALSE; Motor_Abajo_2 := FALSE; END_IF;
(* Network 70 *)
_p58 := S1_2 AND Baja2_21 AND Marcha2;
IF _p58 THEN Marcha2 := FALSE; Baja2_21 := FALSE; Motor_Abajo_2 := FALSE; END_IF;
(* Network 71 *)
_p59 := S3_2 AND Sube2_23 AND Marcha2;
IF _p59 THEN Marcha2 := FALSE; Sube2_23 := FALSE; Motor_Abajo_2 := FALSE; END_IF;
(* Network 72 *)
_p60 := S0_2 AND Baja2_30 AND Marcha2;
IF _p60 THEN Marcha2 := FALSE; Baja2_30 := FALSE; Motor_Abajo_2 := FALSE; END_IF;
(* Network 73 *)
_p61 := S1_2 AND Baja2_31 AND Marcha2;
IF _p61 THEN Marcha2 := FALSE; Baja2_31 := FALSE; Motor_Abajo_2 := FALSE; END_IF;
(* Network 74 *)
_p62 := S2_2 AND Baja2_32 AND Marcha2;
IF _p62 THEN Marcha2 := FALSE; Baja2_32 := FALSE; Motor_Abajo_2 := FALSE; END_IF;
(* Network 75 *)
FIN:
FIN := TRUE;
END_PROGRAM

(* Visualisation Ascensor
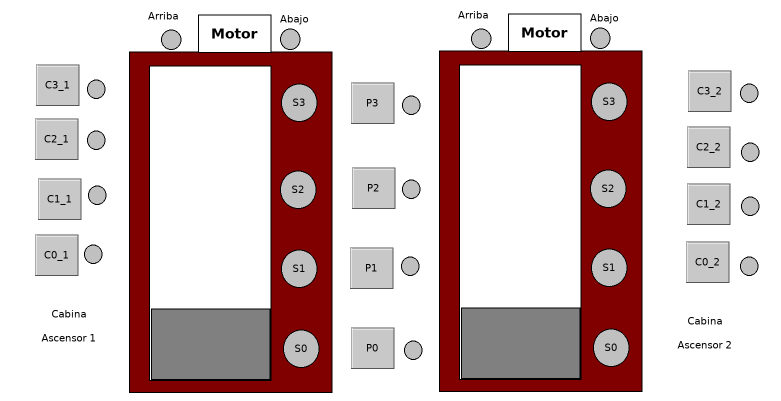
ellipse at (285,341)-(321,379): text "S0"; alarm colour if S0_1
ellipse at (283,261)-(319,299): text "S1"; alarm colour if S1_1
ellipse at (282,182)-(318,220): text "S2"; alarm colour if S2_1
ellipse at (283,95)-(319,133): text "S3"; alarm colour if S3_1
rounded rectangle at (153,320)-(272,391): y offset Movimiento1.pos1
button at (353,339)-(396,380): text "P0"; taps P0
button at (352,259)-(395,300): text "P1"; taps P1
button at (354,179)-(397,220): text "P2"; taps P2
button at (353,94)-(396,135): text "P3"; taps P3
rectangle at (200,26)-(273,64): text "Motor"
ellipse at (163,41)-(183,61): alarm colour if Motor_arriba_1
ellipse at (282,40)-(302,61): alarm colour if Motor_abajo_1
rectangle at (138,18)-(193,37): text "Arriba"
rectangle at (269,21)-(324,40): text "Abajo"
ellipse at (595,340)-(631,378): text "S0"; alarm colour if S0_2
ellipse at (593,260)-(629,298): text "S1"; alarm colour if S1_2
ellipse at (592,181)-(628,219): text "S2"; alarm colour if S2_2
ellipse at (593,94)-(629,132): text "S3"; alarm colour if S3_2
rounded rectangle at (463,319)-(582,390): y offset Movimiento2.pos2
rectangle at (510,25)-(583,63): text "Motor"
ellipse at (473,40)-(493,60): alarm colour if Motor_arriba_2
ellipse at (592,39)-(612,60): alarm colour if Motor_abajo_2
rectangle at (448,17)-(503,36): text "Arriba"
rectangle at (579,20)-(634,39): text "Abajo"
button at (37,246)-(80,287): text "C0_1"; taps C0_1
button at (40,190)-(83,231): text "C1_1"; taps C1_1
button at (37,130)-(80,171): text "C2_1"; taps C2_1
button at (38,76)-(81,117): text "C3_1"; taps C3_1
rectangle at (28,305)-(114,346): text "Cabina"
rectangle at (28,329)-(114,370): text "Ascensor 1"
button at (688,253)-(731,294): text "C0_2"; taps C0_2
button at (689,195)-(732,236): text "C1_2"; taps C1_2
button at (689,138)-(732,179): text "C2_2"; taps C2_2
button at (690,82)-(733,123): text "C3_2"; taps C3_2
rectangle at (664,312)-(750,353): text "Cabina"
rectangle at (664,336)-(750,377): text "Ascensor 2"
ellipse at (89,91)-(107,110): alarm colour if LuzC3_1
ellipse at (89,142)-(107,161): alarm colour if LuzC2_1
ellipse at (90,197)-(108,216): alarm colour if LuzC1_1
ellipse at (86,256)-(104,275): alarm colour if LuzC0_1
ellipse at (404,107)-(422,126): alarm colour if LuzP3
ellipse at (404,191)-(422,210): alarm colour if LuzP2
ellipse at (403,268)-(421,287): alarm colour if LuzP1
ellipse at (406,352)-(424,371): alarm colour if LuzP0
ellipse at (742,95)-(760,114): alarm colour if LuzC3_2
ellipse at (743,154)-(761,173): alarm colour if LuzC2_2
ellipse at (743,208)-(761,227): alarm colour if LuzC1_2
ellipse at (742,268)-(760,287): alarm colour if LuzC0_2
6 more shapes without text or variables
*)
